FUNCTION_BLOCK Q_StringValue (* Command Change String Value ( Part 6 - F.24 ) *)
  (* Standard: ISO 11783-6; Description: Copyright (c) 2022 HR Agrartechnik GmbH This program and the accompanying materials are made available under the terms of the Eclipse Public License 2.0 which is available at https://www.eclipse.org/legal/epl-2.0/ SPDX-License-Identifier: EPL-2.0 see Description Tab *)
  (* Version 1.0, 2022-07-08, Franz Höpfinger, HR Agrartechnik GmbH *)
  PACKAGE isobus::UT::Q;
  IMPORT isobus::UT::Q::const::IDs::ID_NULL;
  (* Documentation:
  Command Change String Value with command buffer reference ( Part 6 - F.24 )
   This command sends a string to the VT. If the ObjectID is already in the command FIFO then the value of this FIFO entry is updated. The length of the string including '\0' may not be longer than the define ISO_VTC_CMD_STR_MAX_LENGTH. Take care that '\0' is trailed.
   Data length / Transport Protocol (F.24): The Change String Value command has a variable data length (command frame: bytes 2–3 Object ID, bytes 4–5 number of string bytes, bytes 6–n string value). Strings that fit into a single CAN message are sent directly; longer strings are transmitted using the ISO 11783 transport protocol. Per Annex F.24 the transferred string may be shorter than the target object's length attribute — the VT pads it with space characters — but the number of bytes transferred shall not exceed the target object's length attribute.
   Valid Object IDs
   A string value Object ID is valid if it falls within one of the following ISO 11783-6 ID ranges:
    - InputStringField: 8000 – 8999
   - OutputStringField: 11000 – 11999
   - StringVariable: 22000 – 22999
   - InputAttributesObject: 26000 – 26999
    ID_NULL (65535) is not a command target but can be used in INIT to deactivate the FB. Any ID outside these ranges is invalid for commanding.
   Activate / Deactivate
   The FB is deactivated by default. It becomes active when INIT provides a valid string value Object ID. Sending INIT with ID_NULL (65535) deactivates the FB again. This toggle can be repeated arbitrarily.
    - INIT + ID_NULL (65535): FB deactivated, STATUS="DEACTIVATED", s16result=VT_E_DEACTIVATED (-40)
   - INIT + valid string value ID: FB activated, STATUS="initialized", s16result=VT_E_NO_ERR (0). If a REQ was buffered before, it is executed immediately.
   - INIT + invalid ID: STATUS="ERROR: Invalid Object ID (not a string value object)", s16result=VT_E_INVALID_OBJECT_ID (-132)
    REQ Handling
    - REQ before any INIT: Buffered, STATUS="Buffered: INIT not yet completed", s16result=VT_E_NOT_READY (-131)
   - REQ while deactivated (INIT came with NULL or invalid ID): STATUS shows the actual deactivation reason, s16result=VT_E_DEACTIVATED (-40) or VT_E_INVALID_OBJECT_ID (-132)
   - REQ while active: Command sent to VT, result reflected in CNF
    param[in] {objectId, iso_u16}
   Object ID. Use ID_NULL (65535) to deactivate the FB. Use a valid string value object ID to activate.
   param[in] {string[], const uint8_t[] }
   Pointer to string
   Return Values (s16result):
   int16_t
    - VT_E_NO_ERR (0) - OK
   - VT_E_DEACTIVATED (-40) - FB deactivated (INIT received with ID_NULL)
   - VT_E_INVALID_OBJECT_ID (-132) - Object ID is invalid (not a string value object)
   - VT_E_NOT_READY (-131) - Buffered: INIT not yet completed
   - VT_E_OVERFLOW (-6) - buffer overflow
   - VT_E_NOACT (-8) - Command not possible in current state
   - VT_E_NO_INSTANCE (-21) - No VT client available
   - VT_E_ISO_INSTANCE_INVALID (-129) - Identifier for instance (connection) invalid
   - VT_E_NOT_ALIVE (-130) - Identifier for instance valid, but VT Dead.
    Instanz-Eindeutigkeit (Instance Uniqueness)
   Dieser Baustein erfordert Instanz-Eindeutigkeit bezüglich u16ObjId. Es darf im gesamten Programm nur eine Instanz von Q_StringValue für dieselbe Ziel-Objekt-ID existieren. Eine zweite Instanz auf dieselbe Objekt-ID wird bei INIT deaktiviert (STATUS = "This objID is already in use").
  *)
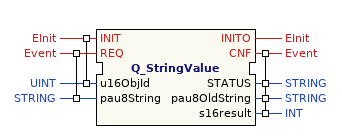
  EVENT_INPUT
    INIT : EInit WITH u16ObjId; (* Service Initialization *)
    REQ WITH pau8String; (* Service Request *)
  END_EVENT
  EVENT_OUTPUT
    INITO : EInit; (* Initialization Confirm *)
    CNF WITH STATUS, pau8OldString, s16result; (* Confirmation of Requested Service *)
  END_EVENT
  VAR_INPUT
    u16ObjId : UINT := ID_NULL; (* Object ID *)
    pau8String : STRING; (* Pointer to string *)
  END_VAR
  VAR_OUTPUT
    STATUS : STRING; (* Service Status *)
    pau8OldString : STRING; (* Old pointer to string *)
    s16result : INT; (* retval see description *)
  END_VAR
END_FUNCTION_BLOCK
